TYPE E_VFS :
(

	At_Vac,
	Triggered,
	Vac_Fault,
	Cls_Timeout,
	Opn_Timeout

);
END_TYPE

(* stored: Version 1.1.0.1, ProductVersion 3.1.4022.18
   DUT E_VFS: Id {4b210349-830f-473c-9f5a-85821adbefb7} *)
